// TIA Portal V17 export
// export: Created 2024-06-19T09:47:15.0835724Z, ExportSetting WithDefaults, DisplayName Totally Integrated Automation Portal, DisplayVersion V17, DisplayName TIA Portal Openness, DisplayVersion V17, DisplayName TIA Portal Version Control Interface, DisplayVersion V17, DisplayName STEP 7 Professional, DisplayVersion V17, DisplayName STEP 7 Safety, DisplayVersion V17, DisplayName WinCC Professional, DisplayVersion V17
VAR_GLOBAL   // PLC tag table "St3_Out"
   IO_Ouverture_TrappeEntree AT %Q1.6 : Bool;   // Ouverture : Trappe d'entrée
   IO_Fermeture_TrappeEntree AT %Q1.7 : Bool;   // Fermeture : Trappe de sortie
   IO_Ouverture_TrappeSortie AT %Q2.0 : Bool;   // Ouverture : Trappe de sortie
   IO_Fermeture_TrappeSortie AT %Q2.1 : Bool;   // Fermeture : Trappe de sortie
   IO_Ouverture_Obturateur AT %Q2.2 : Bool;   // Ouverture : Obturateur
   IO_Fermeture_Obturateur AT %Q2.3 : Bool;   // Fermeture : Obturateur
   IO_Femerture_PorteRX AT %Q2.4 : Bool;   // Ouverte : Porte RX (Homme)
   IO_Ouverture_PorteRX AT %Q2.5 : Bool;   // Fermeture : Porte RX (Homme)
END_VAR
